{attribute 'linkalways'} 
{attribute 'no_explicit_call' := 'This FB is a CLASS and must be accessed using methods or properties'}
{attribute 'enable_dynamic_creation'}
FUNCTION_BLOCK _BOOL EXTENDS DatatypeBase
VAR
	localData : BOOL;
	activeData : REFERENCE TO BOOL REF= localData;
END_VAR

PROPERTY PUBLIC Address : PVOID
GET
Address := ADR(activeData);
END_GET
END_PROPERTY

METHOD PUBLIC ClearReference
VAR_INPUT
END_VAR
activeData REF= localData;
END_METHOD

METHOD PUBLIC Clone : I_Datatype
VAR
    pClone : POINTER TO _BOOL;
END_VAR
pClone := __NEW(_BOOL(InitialValue := Value));
Clone := pClone^;
END_METHOD

METHOD FB_init : BOOL
VAR_INPUT
	bInitRetains : BOOL; // if TRUE, the retain variables are initialized (warm start / cold start)
	bInCopyCode : BOOL;  // if TRUE, the instance afterwards gets moved into the copy code (online change)
	InitialValue : BOOL;
END_VAR
localData := InitialValue;
END_METHOD

METHOD PUBLIC MakeReferenceTo
VAR_INPUT
	ReferenceTarget : REFERENCE TO BOOL;
END_VAR
activeData REF= ReferenceTarget;
END_METHOD

METHOD PUBLIC SerializeWith
VAR_INPUT
	Serializer : I_Serializer;
END_VAR
Serializer.AddBool(activeData);
END_METHOD

PROPERTY PUBLIC Size : UDINT
GET
Size := SIZEOF(activeData);
END_GET
END_PROPERTY

METHOD TryDeserializeFrom : BOOL
VAR_INPUT
	Deserializer : I_Deserializer;
	Feedback : I_DeserializerFeedback;
END_VAR
TryDeserializeFrom := Deserializer.TryGetBool(activeData, Feedback);
END_METHOD

METHOD TryMakeReferenceTo : BOOL
VAR_INPUT
	Target : I_Datatype;
END_VAR
VAR
	pTargetData : POINTER TO BOOL;
END_VAR
IF NOT (Target.TypeName = TypeName) THEN
	RETURN;
END_IF

pTargetData := Target.Address;
activeData REF= pTargetData^;
TryMakeReferenceTo := TRUE;
END_METHOD

PROPERTY PUBLIC TypeName : T_MAXSTRING
GET
TypeName := 'BOOL';
END_GET
END_PROPERTY

PROPERTY PUBLIC Value : REFERENCE TO BOOL
GET
Value REF= activeData;
END_GET
END_PROPERTY

END_FUNCTION_BLOCK

(* stored: Version 1.1.0.1, ProductVersion 3.1.4024.12
   POU _BOOL: Id {42267804-8b15-4f6d-a49b-60c586fde027}, SpecialFunc None
   Folder Constructor: Id {eb40a9e2-d3c8-480b-9f56-3891dcc1f972}
   Property Address: Id {73b368c2-6a1f-4a53-a313-ddeab6ad9073}
   Get Get: Id {67fabb13-fa29-435a-a556-5c946fe19c14}
   Method ClearReference: Id {6d42bdb2-3dbf-4ec6-b688-c729e0abaafa}
   Method Clone: Id {1d1d405f-2859-4fcd-b93c-4a3436f06657}
   Method FB_init: Id {5c024a99-fd8c-4bd3-b4dd-6f5b63b8240c}
   Method MakeReferenceTo: Id {8ac2c2a8-ffe1-41a7-b9a9-fa33a9ad17e7}
   Method SerializeWith: Id {e252c071-95f1-4b1e-a58d-3da5a6b740b6}
   Property Size: Id {b24fd1d1-242c-4f57-8e7a-9bc96dac0ccc}
   Get Get: Id {77056fbe-c14c-40b4-a63a-8db7499bb1f5}
   Method TryDeserializeFrom: Id {1551da21-3487-43a3-8978-847ba01e0c6b}
   Method TryMakeReferenceTo: Id {317170ab-97cf-4198-a0e1-73cfcc6da7b2}
   Property TypeName: Id {32c910a2-3bd6-40dd-9e54-611ce6d5c2c8}
   Get Get: Id {bf4cb1dc-e00a-40d0-99e7-195ebd037272}
   Property Value: Id {64e511bc-d09b-4bb4-ae2d-13ddc41e673a}
   Get Get: Id {bce68bc9-4e3f-4958-b5c1-cd9cc9d6216b} *)
